TYPE HMIXTSMoverHelper_typ :
STRUCT
	BallImgVisibility:			BOOL;
	BallRejectImgVisibility:	BOOL;
	MoverTextVisibility: 		BOOL;
	MoverText: 					STRING;
END_STRUCT
END_TYPE

(* stored: Version 1.1.0.1, ProductVersion 3.1.4024.12
   DUT HMIXTSMoverHelper_typ: Id {3e490a70-6328-0a90-3608-650dbf2daa58} *)
